// TwinCAT 3 PLC project ExternControl
// ProgramVersion: 3.1.4026.19
// libraries:
//   Tc2_Standard, * (Beckhoff Automation GmbH)
//   Tc2_System, * (Beckhoff Automation GmbH)
//   Tc2_Utilities, * (Beckhoff Automation GmbH)
//   VisuDialogs, * (System)
//   VisuDialogs
// project tree:
//   APPLICATION/ fb_Simulation.TcPOU (not stored), GVL_APPLICATION.TcGVL (not stored), MAIN_APP.TcPOU (not stored)
//   APPLICATION/_types/ E_PROCESS_CHECK.TcDUT (not stored), E_PROCESS_CTRL.TcDUT (not stored), E_PROCESS_STATE.TcDUT (not stored), ST_PROCESS_CTRL.TcDUT (not stored), ST_PROCESS_STATE.TcDUT (not stored), T_PROCESS.TcDUT (not stored)
//   APPLICATION/_types/fb_Instance/ E_INSTANCE_CHECK.TcDUT (not stored), E_INSTANCE_STATE.TcDUT (not stored), fb_Instance.TcPOU (not stored)
//   APPLICATION/_types/LinkedList/ fb_Process_LinkedListCtrl.TcPOU (not stored), I_Process_LinkedList.TcIO, ST_PROCESS_DATA.TcDUT (not stored), ST_PROCESS_LIST_RESULT.TcDUT (not stored)
//   / GlobalTextList.TcGTLO (not stored), MAIN.TcPOU, PlcTask.TcTTO (not stored), Visualization Manager.TcVMO (not stored)
//   MAPPING/ MAPPING_in.TcPOU, MAPPING_out.TcPOU
//   MAPPING/_types/ U_APP_CTRL.TcDUT (not stored), U_APP_STATE.TcDUT, U_INSTANCE_CTRL.TcDUT (not stored), U_INSTANCE_STATE.TcDUT (not stored), U_MOVER_CTRL.TcDUT, U_MOVER_INFO.TcDUT (not stored), U_MOVER_STATE.TcDUT (not stored), U_MOVE_DATA.TcDUT, U_TICKET_LIST_CTRL.TcDUT (not stored), U_TICKET_LIST_DATA_INPUT.TcDUT (not stored), U_TICKET_LIST_DATA_OUTPUT.TcDUT (not stored), U_TICKET_LIST_STATE.TcDUT, U_XTS_STATION_CTRL.TcDUT (not stored), U_XTS_STATION_STATE.TcDUT (not stored), U_XTS_TRANSPORT_CTRL.TcDUT (not stored), U_XTS_TRANSPORT_STATE.TcDUT (not stored)
//   MSG/ fb_LocalTime.TcPOU (not stored), fb_MessageData.TcPOU, fb_MessageDataCtrl.TcPOU (not stored), f_MessageSet.TcPOU (not stored), GVL_MSG.TcGVL, I_MessageData.TcIO
//   MSG/types/ e_Device.TcDUT (not stored), E_MessageType.TcDUT (not stored), E_MESSAGE_BATCH.TcDUT, E_MESSAGE_CHECK.TcDUT, E_MESSAGE_CTRL.TcDUT (not stored), E_MESSAGE_FLOW.TcDUT (not stored), E_MESSAGE_STATE.TcDUT (not stored), e_Subdevice.TcDUT (not stored), ST_Message.TcDUT (not stored), ST_MESSAGE_CTRL.TcDUT (not stored), ST_MESSAGE_STATE.TcDUT, TL_E_MESSAGETYPE.TcTLO (not stored)
//   XTS/CaGroup/types/ E_CA_GROUP_STATE.TcDUT (not stored), E_GROUP_CHECK.TcDUT (not stored), ST_GROUP_INFO.TcDUT (not stored)
//   XTS/ GVL_XTS.TcGVL, XTS_Parameter.TcGVL (not stored)
//   XTS/Mover/types/ E_MOVER_CTRL.TcDUT, E_MOVER_STATE.TcDUT (not stored), ST_GEAR_DATA.TcDUT (not stored), ST_MOVER_CTRL.TcDUT (not stored), ST_MOVER_INFO.TcDUT (not stored), ST_MOVER_STATE.TcDUT (not stored), ST_MOVE_DATA.TcDUT
//   XTS/Xpu/types/ E_XPU_CHECK.TcDUT (not stored), E_XPU_CTRL.TcDUT (not stored), E_XPU_INIT.TcDUT (not stored), E_XPU_STATE.TcDUT (not stored), ST_XPU_CTRL.TcDUT, ST_XPU_INFO.TcDUT (not stored), ST_XPU_STATE.TcDUT (not stored)
//   XTS/XtsStation/_types/ E_STATION_CTRL.TcDUT (not stored), E_STATION_GEAR_DISTANCE_AXIS.TcDUT (not stored), E_STATION_STATE.TcDUT (not stored), E_STATION_TYPE.TcDUT, ST_STATION_CTRL.TcDUT (not stored), ST_STATION_GEAR_PARAMETER.TcDUT, ST_STATION_LIST_RESULT.TcDUT (not stored), ST_STATION_MOVER_DATA.TcDUT (not stored), ST_STATION_PARAMETER.TcDUT (not stored), ST_STATION_STATE.TcDUT (not stored), T_NEST_OFFSET.TcDUT (not stored)
//   XTS/XtsTransportUnit/types/ E_XTS_TRANSPORT_CHECK.TcDUT (not stored), E_XTS_TRANSPORT_CTRL.TcDUT (not stored), E_XTS_TRANSPORT_STATE.TcDUT (not stored), ST_XTS_TRANSPORT_CTRL.TcDUT (not stored), ST_XTS_TRANSPORT_STATE.TcDUT (not stored)
//   XTS/_types/ E_PROGRESS.TcDUT (not stored), f_GetProgress.TcPOU (not stored), f_GetState.TcPOU
//   XTS/_Visualization/ GROUP_VISU.TcVIS, MOVER_VISU.TcVIS (not stored), STATION_VISU.TcVIS (not stored), XPU_VISU.TcVIS (not stored), XTS_TRANSPORT.TcVIS (not stored)
//   XTS/_Visualization/textlists/ TL_E_CTRL_MOVER.TcTLO, TL_E_CTRL_STATION.TcTLO (not stored), TL_E_CTRL_TRANSPORT.TcTLO (not stored), TL_E_CTRL_XPU.TcTLO (not stored)
//   XTS/_Visualization/types/ ST_XPU_STRINGS.TcDUT
// (motion and I/O tree: see PLC project xtstransport)
// real-time tasks:
//   TASK XTS Task 1: cycle T#250us, priority 1, ADS port 350
//   TASK PlcTask: cycle T#2ms, priority 15, ADS port 351
//   TASK Job Task: cycle default, priority 32
// variable links:
//   ExternControl/ExternControl Instance <-> XtsTransport/XtsTransport Instance
//     PlcTask Inputs/MAPPING_in.MoverInfo.byInfo <-> PlcTask Outputs/MAPPING_out.MoverInfo.byInfo
//     PlcTask Inputs/MAPPING_in.MoverState.byState <-> PlcTask Outputs/MAPPING_out.MoverState.byState
//     PlcTask Inputs/MAPPING_in.TransportState.byState <-> PlcTask Outputs/MAPPING_out.TransportState.byState
//     PlcTask Outputs/MAPPING_out.MoveData.byData <-> PlcTask Inputs/MAPPING_in.MoveData.byData
//     PlcTask Outputs/MAPPING_out.MoverControl.byCtrl <-> PlcTask Inputs/MAPPING_in.MoverCtrl.byCtrl
//     PlcTask Outputs/MAPPING_out.TransportControl.byCtrl <-> PlcTask Inputs/MAPPING_in.TransportControl.byCtrl

// ---- MAPPING/_types/U_APP_STATE.TcDUT
TYPE U_APP_STATE :
UNION
  stState             : ST_APP_STATE;
  byState   AT %i*    : ARRAY[1..SIZEOF(ST_APP_STATE)] OF BYTE;
END_UNION
END_TYPE

// ---- MAPPING/_types/U_MOVER_CTRL.TcDUT
TYPE U_MOVER_CTRL :
UNION
  stCtrl              : ARRAY[1..MAX_MOVER] OF ST_MOVER_CTRL;

  byCtrl    AT %Q*    : ARRAY[1..MAX_MOVER] OF
                        ARRAY[1..SIZEOF(ST_MOVER_CTRL)] OF BYTE;
END_UNION
END_TYPE

// ---- MAPPING/_types/U_MOVE_DATA.TcDUT
TYPE U_MOVE_DATA :
UNION
  stData              : ARRAY[1..MAX_MOVER] OF ST_MOVE_DATA;

  byData    AT %Q*    : ARRAY[1..MAX_MOVER] OF
                        ARRAY[1..SIZEOF(ST_MOVE_DATA)] OF BYTE;
END_UNION
END_TYPE

// ---- MAPPING/_types/U_TICKET_LIST_STATE.TcDUT
TYPE U_TICKET_LIST_STATE :
UNION
  stState             : ST_LIST_STATE;
  byState   AT %I*    : ARRAY[1..SIZEOF(ST_LIST_STATE)] OF BYTE;
END_UNION
END_TYPE

// ---- MSG/types/E_MESSAGE_BATCH.TcDUT
{attribute 'qualified_only'}
{attribute 'strict'}
{attribute 'to_string'}
TYPE E_MESSAGE_BATCH :
(
	MSG_BATCH_NULL,
  MSG_BATCH_JOB_STARTED,
  MSG_BATCH_NEXT_IN_JOB,
  MSG_BATCH_JOB_DONE
)UINT;
END_TYPE

// ---- MSG/types/E_MESSAGE_CHECK.TcDUT
{attribute 'qualified_only'}
{attribute 'strict'}
{attribute 'to_string'}
TYPE E_MESSAGE_CHECK :
(
  // 9000 --> here comes your error
  MSG_CHECK_INVALID_POINTER             := 9000,
  MSG_CHECK_INVALID_POINTER_TIME,
  MSG_CHECK_INVALID_POINTER_LIST,
  MSG_CHECK_INVALID_POINTER_MSG_IDX,
  MSG_CHECK_INVALID_POINTER_ERR_IDX,
  MSG_CHECK_INVALID_POINTER_ROOT_FILE,
  MSG_CHECK_INVALID_POINTER_ROOT_DIR,
  MSG_CHECK_INVALID_POINTER_CTRL,
  MSG_CHECK_INVALID_POINTER_STATE,

  // 10000 --> here comes your man
  MSG_CHECK_DONE                        := 10000
)UINT;
END_TYPE

// ---- MSG/types/ST_MESSAGE_STATE.TcDUT
TYPE ST_MESSAGE_STATE :
STRUCT
  State         : E_MESSAGE_STATE;  // as always... combined value of Cmd equivalent and e_progress
END_STRUCT
END_TYPE

// ---- XTS/Mover/types/E_MOVER_CTRL.TcDUT
{attribute 'qualified_only'}
{attribute 'strict'}
{attribute 'to_string'}
TYPE E_MOVER_CTRL :
(
  MOVER_NULL,               // initial value at startup, used for change of order or retrigger
  MOVER_ENABLE,             // sets MC_Power.Enable
  MOVER_DISABLE,            // removes MC_Power.Enable
  MOVER_MOVE_TO_POS,        // modulo absolute positioning with MC_MoveAbsolute, InTargetPosition check
  MOVER_MOVE_TO_POS_CA,     // modulo absolute positioning with MC_MoveAbsoluteCA, InTargetPosition check
  MOVER_SEND_TO_POS_CA,     // modulo absolute positioning with MC_MoveAbsoluteCA, done after moving ReleaseDistance
  MOVER_HALT,               // halts mover; by use of MC_Halt mover is set passive in CA group
  MOVER_GEAR_IN,            // GearIn for mover in standstill

  MOVER_GEAR_IN_POS_CA,     // GearInPosCA of mover; when FB_GearInPosCa is InSync --> order is done; check SyncDistance yourself and release mover with e_mover_order.mover_SendToPos
  MOVER_GEAR_OUT,           // gear out for mover
  MOVER_RESET,              // MC_RESET for mover
  MOVER_MOVE_TO_POS_ABS    // absolute positioning with MC_MoveAbsolute, InTargetPosition check
)UINT;
END_TYPE

// ---- XTS/Mover/types/ST_MOVE_DATA.TcDUT
{attribute 'pack_mode' := '2'}
TYPE ST_MOVE_DATA :
STRUCT
  // HAUD 2024 03 14
  // some init data added for example
  rPos            : LREAL :=   2275.0;
  rVelo           : LREAL :=    500.0;
  rAcc            : LREAL :=   5000.0;
  rJerk           : LREAL := 500000.0;
  rGap            : LREAL :=    100.0;
  rOverride       : LREAL :=    100.0;
  rDelta          : LREAL :=      0.05;
  rDistance       : LREAL :=     25.0;
END_STRUCT
END_TYPE

// ---- XTS/Xpu/types/ST_XPU_CTRL.TcDUT
{attribute 'pack_mode' := '2'}
TYPE ST_XPU_CTRL :
STRUCT
  Cmd             : E_XPU_CTRL;
END_STRUCT
END_TYPE

// ---- XTS/XtsStation/_types/E_STATION_TYPE.TcDUT
{attribute 'qualified_only'}
{attribute 'strict'}
{attribute 'to_string'}
TYPE E_STATION_TYPE :
(
	INVALID,
  STATION_PROCESS,      // default station with/without process
  STATION_GEAR_IN_POS   // GearInPos station for flying saw with MasterAxis
)USINT;
END_TYPE

// ---- XTS/XtsStation/_types/ST_STATION_GEAR_PARAMETER.TcDUT
TYPE ST_STATION_GEAR_PARAMETER :
STRUCT
  eDistance           : E_STATION_GEAR_DISTANCE_AXIS; // follow which leader?
  rSyncDistance       : LREAL := 100.0;               // synchrone distance while the mover is geared in
  rMinDistanceToSync  : LREAL := 100.0;               // minimum distance for mover to get nSync with the Master
END_STRUCT
END_TYPE

// ---- XTS/_Visualization/types/ST_XPU_STRINGS.TcDUT
TYPE ST_XPU_STRINGS :
STRUCT
  sXpuState       ,
  sXpuResult      ,
  sXpuCyclicCheck ,
  sXpuOpMode      ,
  sXpuMoverId_DetectionMode,
  sXpuMoverPosAssignement : STRING(30) := 'NULL';
END_STRUCT
END_TYPE

// ---- MSG/GVL_MSG.TcGVL
{attribute 'qualified_only'}
VAR_GLOBAL CONSTANT
  //-----------------------------------------------------------------------------
  // file paths for message system
  //  - compiler define option WIN switches to Windows file paths
  //-----------------------------------------------------------------------------
{IF defined (WIN)}
  {info 'WIN folders'}
  LOG_DIR               : STRING  := 'C:\TwinCAT\#MsgFiles\'; // delimiter at the end is mandatory!!
{ELSE}
  {info 'BSD folders'}
  LOG_DIR               : STRING  := '/usr/local/etc/TwinCAT/#MsgFiles/'; // delimiter at the end is mandatory!!
{END_IF}

  LOG_FILE              : STRING  := 'MSG_XtsTransport_';
  LOG_FILE_APP          : STRING  := 'MSG_Application_';
  LOG_FILE_METRIC       : STRING  := 'MSG_XtsTransportMetrics_';

  MAX_MESSAGE           : UINT    := 2000; // max entry in message list
END_VAR
VAR_GLOBAL
  //-----------------------------------------------------------------------------
  // Message System
  //  - Everybody uses f_MessageSet(ST_Message)
  //    - DECISION WHICH LIST IS MADE IN f_MessageSet !!
  //    - which list to use is determined by e_Device in your message
  //
  //  - MessageData instances are self sufficient and need only 
  //    datafield assignment for correct data-flow
  //
  //
  //-----------------------------------------------------------------------------
  //-----------------------------------------------------------------------------
  //-----------------------------------------------------------------------------
  // (ST_Message.eDevice := e_Device.Application)
  //----------------------------------------------------------------------------- 
  ApplicationMessageData          : fb_MessageDataCtrl;
  ApplicationMessageCtrl          : st_message_ctrl;
  ApplicationMessageState         : st_message_state;

  ApplicationMessages             : ARRAY[1..MAX_MESSAGE] OF ST_Message;
  MessageApplicationIndex         : UINT := 0; // message index for higher layers (grouping, Instances, etc.)
  MessageApplicationError         : UINT := 0; // error counter for higher learning
  //-----------------------------------------------------------------------------
  //-----------------------------------------------------------------------------
  // (ST_Message.eDevice := from Device_Null to XfcAxis)
  //-----------------------------------------------------------------------------
  TransportMessageData            : fb_MessageDataCtrl;
  TransportMessageCtrl            : st_message_ctrl;
  TransportMessageState           : st_message_state;

  TransportMessages               : ARRAY[1..MAX_MESSAGE] OF ST_Message;
  MessageTransportIndex           : UINT := 0; // message index for base layer
  MessageTransportError           : UINT := 0; // error counter for base layer
  //-----------------------------------------------------------------------------
  //-----------------------------------------------------------------------------
  // (ST_Message.eDevice := e_Device.Metrics)
  //-----------------------------------------------------------------------------
  MetricsMessageData              : fb_MessageDataCtrl;
  MetricsMessageCtrl              : st_message_ctrl;
  MetricsMessageState             : st_message_state;

  MetricsMessages                 : ARRAY[1..MAX_MESSAGE] OF ST_Message;
  MessageMetricsIndex             : UINT := 0; // message index for metrics data
  MessageMetricsError             : UINT := 0; // error counter for metrics data
  //-----------------------------------------------------------------------------
  //-----------------------------------------------------------------------------
  // (ST_Message.eDevice := e_Device.ProductData)
  //-----------------------------------------------------------------------------
  ProductMessageData              : fb_MessageDataCtrl;   // This is for you
  ProductMessageCtrl              : st_message_ctrl;
  ProductMessageState             : st_message_state;

  ProductMessages                 : ARRAY[1..MAX_MESSAGE] OF ST_Message;
  MessageProductIndex             : UINT := 0; // message index for your product data
  MessageProductError             : UINT := 0; // error counter for your product data
  //-----------------------------------------------------------------------------
  //-----------------------------------------------------------------------------
  fbLocalTime                     : fb_LocalTime;
  dtLocalTime                     : DT;
  sLocalTime                      : STRING;
  //-----------------------------------------------------------------------------
  //-----------------------------------------------------------------------------
  //-----------------------------------------------------------------------------
  //-----------------------------------------------------------------------------
  MessageLevelXpu                 : E_MessageType;
  MessageLevelStations            : ARRAY[1..MAX_STATION] OF E_MessageType;
  MessageLevelMovers              : ARRAY[1..MAX_MOVER]   OF E_MessageType;

  MessageLevelProcess             : ARRAY[1..MAX_PROCESS] OF E_MessageType;

{IF defined (TEST)}
  {info 'TEST logging enabled'}
  MessageLevel                    : E_MessageType := eMessageinfo; // a lot of messages
{ELSE}
  MessageLevel                    : E_MessageType := eMessageEmpty; // only errors are written into list 
{END_IF}

END_VAR

// ---- XTS/GVL_XTS.TcGVL
{attribute 'qualified_only'}
VAR_GLOBAL
  //---------------------------------------------------------------------------
  // XTS Station
  //  - handshakes mover in station with extern control
  //  - station parameters (positions, gap, dyn. constraints, description...)
//  StationStart        : ST_STATION_PARAMETER;   // Xts transport is sending all mover to this position (CMD_TRANSPORT_START)
//  StationStartIndex   : UINT := 1;              // index of XtsStation where all movers are entered into linked list.

  // station handshaking with mover and extern process
  // station sends mover to target station/WaitPos
  // station adds mover data to LinkedList.AddTail() of target station
//  Station             : ARRAY[1..MAX_STATION] OF fb_StationProcess;
//  StationGearIn       : ARRAY[1..MAX_STATION] OF fb_StationGearInPos;
//
//  StationList         : ARRAY[1..MAX_STATION] OF fb_Station_LinkedList;
//
//  StationQueue        : ARRAY[1..MAX_STATION]    OF 
//                        ARRAY[1..MAX_LIST_NODES] OF ST_STATION_MOVER_DATA;
//
//  // interface for access to List methods
//  StationListItf      : ARRAY[1..MAX_STATION] OF I_Station_LinkedList;
//
//  // interface for access to station methods
//  StationCtrlItf      : ARRAY[1..MAX_STATION] OF I_XtsTransport_Station;

  // ctrl / state datafields for extern control
  StationCtrl         : ARRAY[1..MAX_STATION] OF ST_STATION_CTRL;   // control for extern to write, you can do whatever you want as long as you do as I say
  StationState        : ARRAY[1..MAX_STATION] OF ST_STATION_STATE;  // state for extern to read, this is what I tell you to do

  // station parameter
//  StationParameter    : ARRAY[1..MAX_STATION] OF ST_STATION_PARAMETER; // wherever, whenever you want. Build it and they will come...

  // station GearInPosCA parameter and data structs
//  StationGearParameter: ARRAY[1..MAX_STATION] OF ST_STATION_GEAR_PARAMETER;
//  StationGearData     : ARRAY[1..MAX_STATION] OF ST_GEAR_DATA;

  // static position offsets in stations
//  PositionOffset      : ARRAY[1..MAX_STATION] OF T_NEST_OFFSET; // added to PosStop[] in XtsStation


  //---------------------------------------------------------------------------
  // XTS
  // XTS TransportUnit
  //  - This is ground control
  //  - handles request for XPU, Group, Mover, StartUp, ReStart
//  XtsTransport        : fb_TransportUnit;         // manages members of XTS transport for extern to access

  XtsTransportCtrl    : ST_XTS_TRANSPORT_CTRL;    // control of XTS transport for extern to write
  XtsTransportState   : ST_XTS_TRANSPORT_STATE;   // state   of XTS transport for extern to read


  //---------------------------------------------------------------------------
  // XPU
  // XTS-Utility checks
  // XTS-Utility interfaces for you to use
//  Xpu             : fb_XpuCtrl;

//  XpuCtrl         : ST_XPU_CTRL;
//  XpuState        : ST_XPU_STATE;
//  XpuInfo         : ST_XPU_INFO;
//  XpuModules      : ARRAY[1..MAX_MODULE] OF Tc3_XTS_Utility.ST_InfoDataView;


  //---------------------------------------------------------------------------
  // Collision avoidance group CA
  //
  // - add mover to group
  // - build group
  // - clear group
  // - whereever you may roam, no on will tread on you
//  CaGroup         : FB_CaGroup;                   // cyclic check of CaGroup state and errors; carries methods for handling CaGroup
//  CaGroupItf      : I_XtsTransport_CaGroup;       // Interface used by fb_TransportUnit

  // cyclic mapping to MOTION/Objects/CaGroup 
//  CaGroupRef      : Tc3_McCoordinatedMotion.AXES_GROUP_REF;

  // Info data from CaGroup FB
//  CaGroupInfo     : ST_GROUP_INFO;                // cyclic info about CaGroup for fb_TransportUnit to read
  //---------------------------------------------------------------------------

  //---------------------------------------------------------------------------
  // MC2 encapsulation, CA movement
//  Mover           : ARRAY[1..MAX_MOVER] OF fb_MoverCtrl;    // MC and CA methods for mover; cyclic check for individual command on mover

  MoverCtrl       : ARRAY[1..MAX_MOVER] OF ST_MOVER_CTRL;   // control of individual mover for extern to write
  MoverState      : ARRAY[1..MAX_MOVER] OF ST_MOVER_STATE;  // state   of individual mover for extern to read

//  MoverItf        : ARRAY[1..MAX_MOVER] OF I_XtsTransport_Mover;  // Interface used by fb_TransportUnit

//  LastPosition    : ARRAY[1..MAX_MOVER] OF LREAL;           // on execute of any movement, value is saved here (used by fb_Mover)
//  LastGap         : ARRAY[1..MAX_MOVER] OF LREAL;           // on execute of any movement, value is saved here (used by fb_Mover)

  MoverInfo       : ARRAY[1..MAX_MOVER] OF ST_MOVER_INFO;   // cyclic info about mover for extern to read

  MoveData        : ARRAY[1..MAX_MOVER] OF ST_MOVE_DATA;    // dynamic constraints for move commands
  GearData        : ARRAY[1..MAX_MOVER] OF ST_GEAR_DATA;    // dynamic constraints and positions for GearIn/GearInPosCa
  
  // cyclic mapping to MOTION/Axes
//  AxisRefMover    : ARRAY[1..MAX_MOVER] OF Tc2_MC2.AXIS_REF;
  //---------------------------------------------------------------------------
END_VAR

// ---- APPLICATION/_types/LinkedList/I_Process_LinkedList.TcIO
INTERFACE I_Process_LinkedList

METHOD AddHeadValue : ST_PROCESS_LIST_RESULT
VAR_INPUT
  stData        : ST_PROCESS_DATA;
END_VAR
END_METHOD

METHOD AddTailValue : ST_PROCESS_LIST_RESULT
VAR_INPUT
  stData        : ST_PROCESS_DATA;
END_VAR
END_METHOD

PROPERTY Count : UDINT
GET
END_GET
END_PROPERTY

PROPERTY Data : ARRAY[1..MAX_LIST_NODES] OF ST_PROCESS_DATA
GET
END_GET
END_PROPERTY

PROPERTY Free : UDINT
GET
END_GET
END_PROPERTY

METHOD GetHead : ST_PROCESS_LIST_RESULT
VAR_INPUT
END_VAR
END_METHOD

METHOD InitList : BOOL
END_METHOD

PROPERTY Nodes : ARRAY[0..MAX_LIST_NODES] OF T_LinkedListEntry
GET
END_GET
END_PROPERTY

METHOD RemoveHeadValue : ST_PROCESS_LIST_RESULT
VAR_INPUT
END_VAR
END_METHOD

END_INTERFACE

// ---- MSG/I_MessageData.TcIO
INTERFACE I_MessageData

PROPERTY DirRoot : POINTER to string(255)
SET
END_SET
END_PROPERTY

PROPERTY ErrorIndex : reference to uint
SET
END_SET
END_PROPERTY

PROPERTY FileRoot : pointer to string(255)
SET
END_SET
END_PROPERTY

PROPERTY LocalTime : pointer to DT
SET
END_SET
END_PROPERTY

PROPERTY MessageIndex : reference to uint
SET
END_SET
END_PROPERTY

PROPERTY MsgList : pointer to ARRAY[1..GVL_MSG.MAX_MESSAGE] OF st_message
SET
END_SET
END_PROPERTY

END_INTERFACE

// ---- MAIN.TcPOU
//---------------------------------------------------------------------------------------------------------------
//
//  HAUD 2026.01.16
//
//  - ExternControl
//
//    - placeholder programm for specific implementation of machine logic
//
//---------------------------------------------------------------------------------------------------------------
PROGRAM MAIN
VAR
	bInit 				          : BOOL;
  eInit                   : E_PROGRESS := E_PROGRESS.PROGRESS_DONE; // empty right now, so init is done

  nStation,
	nMover,
  nMoverSelected,
  nStationSelected,
  nStationParameter       : UINT;

  sStationText            : STRING(30);
  stXpuStrings            : ST_XPU_STRINGS;

  eTransportState         : E_XTS_TRANSPORT_STATE;
  eTransportResult        : E_PROGRESS;

  eXpuState               : E_XPU_STATE;
  eXpuResult              : E_PROGRESS;
  eXpuCheck               : E_XPU_CHECK;

  eMoverState             : E_MOVER_STATE;
  eMoverResult            : E_PROGRESS;

  sCaGroupState,
  sTransportState,
  sTransportCheck,
  sTransportResult,
  sMoverState,
  sMoverResult,
  sStationState,
  sStationStateMask,
  sStationCtrlMask        : STRING;

  bStationEnable,
  bStationEnter,
  bStationStart,
  bStationDone,
  bStationOut,
  bStationGone            : BOOL;

  nStn                    : UINT;

  stMsg                   : ST_Message;
  eMsgState               : e_message_state;
  eMsgProgress            : E_PROGRESS;
  eMtrState               : e_message_state;
  eMtrProgress            : E_PROGRESS;

  bGetVariant             : BOOL := TRUE;
  nVariant                : UINT;

  rGap                    : REAL :=     105.0;
  rAcc                    : REAL :=  17_500.0;
  rJerk                   : REAL := 600_000.0;
END_VAR

//############################################################################
//############################################################################
//  /Visualization data	
//############################################################################
VisualizationData();
//############################################################################
//  Visualization data/	
//############################################################################

ACTION VisualizationData:
//############################################################################
//############################################################################
// Visualization data	
//############################################################################
// get enumerations from XPU for visu:	
eTransportState                       := f_GetState   (GVL_XTS.XtsTransportState.State);
eTransportResult                      := f_GetProgress(GVL_XTS.XtsTransportState.State);

eXpuState                             := f_GetState   (GVL_XTS.XtsTransportState.XpuState.State);
eXpuResult                            := f_GetProgress(GVL_XTS.XtsTransportState.XpuState.State);

eXpuCheck                             := GVL_XTS.XtsTransportState.XpuState.Check;

// display xpu state and result in visu
// get strings and info
sCaGroupState                         := TO_STRING(GVL_XTS.XtsTransportState.GroupInfo.CaGroupState);

sTransportState                       := TO_STRING(eTransportState);
sTransportCheck                       := TO_STRING(GVL_XTS.XtsTransportState.Check);
sTransportResult                      := TO_STRING(eTransportResult);

stXpuStrings.sXpuState                := TO_STRING(eXpuState);
stXpuStrings.sXpuResult               := TO_STRING(eXpuResult);
stXpuStrings.sXpuCyclicCheck          := TO_STRING(eXpuCheck);

stXpuStrings.sXpuOpMode               := TO_STRING(GVL_XTS.XtsTransportState.XpuInfo.OperationMode);
stXpuStrings.sXpuMoverId_DetectionMode:= TO_STRING(GVL_XTS.XtsTransportState.XpuInfo.IdDetectionMode);
stXpuStrings.sXpuMoverPosAssignement  := TO_STRING(GVL_XTS.XtsTransportState.XpuInfo.MoverPositionAssignement);

nMoverSelected                        := SEL((nMoverSelected<1), nMoverSelected, 1);
nMoverSelected                        := SEL((nMoverSelected>MAX_MOVER), nMoverSelected, MAX_MOVER);

nStationSelected                      := SEL((nStationSelected<1), nStationSelected, 1);
nStationSelected                      := SEL((nStationSelected>MAX_STATION), nStationSelected, MAX_STATION);

//bStationEnable                        := SEL((GVL_XTS.StationCtrl[nStationSelected].Cmd = E_STATION_CTRL.STATION_ENABLE),        FALSE, TRUE);
//bStationEnter                         := SEL((GVL_XTS.StationCtrl[nStationSelected].Cmd = E_STATION_CTRL.STATION_MOVER_ENTER),   FALSE, TRUE);
//bStationStart                         := SEL((GVL_XTS.StationCtrl[nStationSelected].Cmd = E_STATION_CTRL.STATION_PROCESS_START), FALSE, TRUE);
//bStationDone                          := SEL((GVL_XTS.StationCtrl[nStationSelected].Cmd = E_STATION_CTRL.STATION_PROCESS_DONE),  FALSE, TRUE);
//bStationOut                           := SEL((GVL_XTS.StationCtrl[nStationSelected].Cmd = E_STATION_CTRL.STATION_MOVER_OUT),     FALSE, TRUE);
//bStationGone                          := SEL((GVL_XTS.StationCtrl[nStationSelected].Cmd = E_STATION_CTRL.STATION_MOVER_GONE),    FALSE, TRUE);

eMoverState                           := f_GetState   (GVL_XTS.MoverState[nMoverSelected].State);
eMoverResult                          := f_GetProgress(GVL_XTS.MoverState[nMoverSelected].State);

sMoverState                           := TO_STRING(eMoverState);
sMoverResult                          := TO_STRING(eMoverResult);

//sStationState                         := TO_STRING(GVL_XTS.StationState[nStationSelected].State);
//sStationStateMask                     := Tc2_Utilities.BYTE_TO_BINSTR(GVL_XTS.StationState[nStationSelected].nMask, 8);
//sStationCtrlMask                      := Tc2_Utilities.BYTE_TO_BINSTR(GVL_XTS.StationCtrl[nStationSelected].nMask, 8);

//############################################################################
//############################################################################
END_ACTION

END_PROGRAM

// ---- XTS/_types/f_GetState.TcPOU
// global function to extract state identifier from combined value
FUNCTION f_GetState : uint
VAR_INPUT
  state     : UINT; // combined value of identifier + e_progress
END_VAR
VAR
  _stx      : uint;
END_VAR

_stx          := state MOD E_PROGRESS.PROGRESS_INIT;

IF (_stx = 0)
THEN
  f_GetState  := state;
ELSE
  f_GetState  := _stx;
END_IF

END_FUNCTION

// ---- MAPPING/MAPPING_in.TcPOU
PROGRAM MAPPING_in
VAR
  sMapping          : STRING;
  bFirstCycle       : BOOL := TRUE;



//  TicketListOutput  : U_TICKET_LIST_DATA_OUTPUT;
//  TicketListState   : U_TICKET_LIST_STATE;
//  InstanceState     : U_INSTANCE_STATE;
//  AppState          : U_APP_STATE;
  TransportState    : U_XTS_TRANSPORT_STATE;
  StationState      : U_XTS_STATION_STATE;
  MoverState        : U_MOVER_STATE;
  MoverInfo         : U_MOVER_INFO;

  szTransportState  : ARRAY[1..2] OF UDINT;
  szStationState    : ARRAY[1..2] OF UDINT;
  szMoverState      : ARRAY[1..2] OF UDINT;
  szMoverInfo       : ARRAY[1..2] OF UDINT;

  szAppState        : ARRAY[1..2] OF UDINT;
  szInstanceState   : ARRAY[1..2] OF UDINT;
  szTicketState     : ARRAY[1..2] OF UDINT;
  szTicketData      : ARRAY[1..2] OF UDINT;
END_VAR


IF (bFirstCycle)
THEN
  bFirstCycle           := FALSE;
  
  szTransportState[1]   := SIZEOF(TransportState);
  szTransportState[2]   := SIZEOF(GVL_XTS.XtsTransportState);

  szStationState  [1]   := SIZEOF(StationState);
  szStationState  [2]   := SIZEOF(GVL_XTS.StationState);

  szMoverState    [1]   := SIZEOF(MoverState);
  szMoverState    [2]   := SIZEOF(GVL_XTS.MoverState);

  szMoverInfo     [1]   := SIZEOF(MoverInfo);
  szMoverInfo     [2]   := SIZEOF(GVL_XTS.MoverInfo);


(*
  szAppState[1]       := SIZEOF(AppState);
  szAppState[2]       := SIZEOF(GVL_APPLICATION.AppState);

  szInstanceState[1]  := SIZEOF(InstanceState);
  szInstanceState[2]  := SIZEOF(GVL_APPLICATION.InstanceState);

  szTicketState[1]    := SIZEOF(TicketListState);
  szTicketState[2]    := SIZEOF(GVL_APPLICATION.TicketListState);

  szTicketData[1]     := SIZEOF(TicketListOutput);
  szTicketData[2]     := SIZEOF(GVL_APPLICATION.TicketListDataOutput);
*)
END_IF
(*
//---------------------------------------------------------------------
IF (SIZEOF(TicketListOutput) <> SIZEOF(GVL_APPLICATION.TicketListDataOutput))
THEN
  sMapping  := 'TicketListOutput sizes DO NOT match';
  RETURN;
END_IF
//---------------------------------------------------------------------
IF (SIZEOF(TicketListState) <> SIZEOF(GVL_APPLICATION.TicketListState))
THEN
  sMapping  := 'TicketListState sizes DO NOT match';
  RETURN;
END_IF
//---------------------------------------------------------------------
IF (SIZEOF(InstanceState) <> SIZEOF(GVL_APPLICATION.InstanceState))
THEN
  sMapping  := 'InstanceState sizes DO NOT match';
  RETURN;
END_IF
//---------------------------------------------------------------------
IF (SIZEOF(AppState) <> SIZEOF(GVL_APPLICATION.AppState))
THEN
  sMapping  := 'AppState sizes DO NOT match';
  RETURN;
END_IF
*)
//---------------------------------------------------------------------
IF (SIZEOF(TransportState) <> SIZEOF(GVL_XTS.XtsTransportState))
THEN
  sMapping  := 'TransportState sizes DO NOT match';
  RETURN;
END_IF
//---------------------------------------------------------------------
IF (SIZEOF(StationState) <> SIZEOF(GVL_XTS.StationState))
THEN
  sMapping  := 'StationState sizes DO NOT match';
  RETURN;
END_IF
IF (SIZEOF(MoverState) <> SIZEOF(GVL_XTS.MoverState))
THEN
  sMapping  := 'MoverState sizes DO NOT match';
  RETURN;
END_IF
IF (SIZEOF(MoverInfo) <> SIZEOF(GVL_XTS.MoverInfo))
THEN
  sMapping  := 'MoverInfo sizes DO NOT match';
  RETURN;
END_IF
sMapping    := 'MAPPING ACTIVE';
//-----------------------------------------------------------------------------------------
//       destination,                               source,                size
//-----------------------------------------------------------------------------------------
  memcpy(ADR(GVL_XTS.XtsTransportState),            ADR(TransportState),  SIZEOF(TransportState));
  memcpy(ADR(GVL_XTS.StationState),                 ADR(StationState),    SIZEOF(StationState));
  memcpy(ADR(GVL_XTS.MoverState),                   ADR(MoverState),      SIZEOF(MoverState));
  memcpy(ADR(GVL_XTS.MoverInfo),                    ADR(MoverInfo),       SIZEOF(MoverInfo));

  //memcpy(ADR(GVL_APPLICATION.AppState),             ADR(AppState),         SIZEOF(AppState));
  //GVL_APPLICATION.AppState.AppInit                  := AppSTate.stState.AppInit;

  //memcpy(ADR(GVL_APPLICATION.InstanceState),        ADR(InstanceState),    SIZEOF(InstanceState));
  //memcpy(ADR(GVL_APPLICATION.TicketListState),      ADR(TicketListState),  SIZEOF(TicketListState));
  //memcpy(ADR(GVL_APPLICATION.TicketListDataOutput), ADR(TicketListOutput), SIZEOF(TicketListOutput));
//-----------------------------------------------------------------------------------------
//-----------------------------------------------------------------------------------------

END_PROGRAM

// ---- MAPPING/MAPPING_out.TcPOU
PROGRAM MAPPING_out
VAR
  sMapping          : STRING;

  bFirstCycle       : BOOL := TRUE;

//  TicketListInput   : U_TICKET_LIST_DATA_INPUT;
//  TicketListControl : U_TICKET_LIST_CTRL;
//  InstanceCtrl      : U_INSTANCE_CTRL;
//  AppControl        : U_APP_CTRL;
  TransportControl  : U_XTS_TRANSPORT_CTRL;
  StationControl    : U_XTS_STATION_CTRL;
  MoverControl      : U_MOVER_CTRL;
  MoveData          : U_MOVE_DATA;



  szTransportCtrl   : ARRAY[1..2] OF UDINT;
  szStationControl  : ARRAY[1..2] OF UDINT;
  szMoverControl    : ARRAY[1..2] OF UDINT;
  szMoveData        : ARRAY[1..2] OF UDINT;

  szAppCtrl         : ARRAY[1..2] OF UDINT;
  szInstanceCtrl    : ARRAY[1..2] OF UDINT;
  szTicketCtrl      : ARRAY[1..2] OF UDINT;
  szTicketData      : ARRAY[1..2] OF UDINT;
END_VAR


IF (bFirstCycle)
THEN
  bFirstCycle             := FALSE;

  szTransportCtrl[1]      := SIZEOF(TransportControl);
  szTransportCtrl[2]      := SIZEOF(GVL_XTS.XtsTransportCtrl);

  szStationControl[1]     := SIZEOF(StationControl);
  szStationControl[2]     := SIZEOF(GVL_XTS.StationCtrl);

  szMoverControl[1]       := SIZEOF(MoverControl);
  szMoverControl[2]       := SIZEOF(GVL_XTS.MoverCtrl);

  szMoveData    [1]       := SIZEOF(MoveData);
  szMoveData    [2]       := SIZEOF(GVL_XTS.MoveData);

(*
  szAppCtrl  [1]          := SIZEOF(AppControl);
  szAppCtrl  [2]          := SIZEOF(GVL_APPLICATION.AppControl);

  szInstanceCtrl [1]      := SIZEOF(MAPPING_out.InstanceCtrl);
  szInstanceCtrl [2]      := SIZEOF(MAPPING_out.InstanceCtrl);

  szTicketCtrl[1]         := SIZEOF(TicketListControl);
  szTicketCtrl[2]         := SIZEOF(GVL_APPLICATION.TicketListControl);

  szTicketData[1]         := SIZEOF(TicketListInput);
  szTicketData[2]         := SIZEOF(GVL_APPLICATION.TicketListDataInput);
*)
END_IF
(*
//---------------------------------------------------------------------
IF (SIZEOF(TicketListInput) <> SIZEOF(GVL_APPLICATION.TicketListDataInput))
THEN
  sMapping  := 'TicketListInput sizes DO NOT match';
  RETURN;
END_IF
//---------------------------------------------------------------------
IF (SIZEOF(TicketListControl) <> SIZEOF(GVL_APPLICATION.TicketListControl))
THEN
  sMapping  := 'TicketListControl sizes DO NOT match';
  RETURN;
END_IF
//---------------------------------------------------------------------
IF (SIZEOF(InstanceCtrl) <> SIZEOF(GVL_APPLICATION.InstanceCtrl))
THEN
  sMapping  := 'InstanceCtrl sizes DO NOT match';
  RETURN;
END_IF
//---------------------------------------------------------------------
IF (SIZEOF(AppControl) <> SIZEOF(GVL_APPLICATION.AppControl))
THEN
  sMapping  := 'AppControl sizes DO NOT match';
  RETURN;
END_IF
*)
//---------------------------------------------------------------------
IF (SIZEOF(TransportControl) <> SIZEOF(GVL_XTS.XtsTransportCtrl))
THEN
  sMapping  := 'TransportControl sizes DO NOT match';
  RETURN;
END_IF
IF (SIZEOF(StationControl) <> SIZEOF(GVL_XTS.StationCtrl))
THEN
  sMapping  := 'StationControl sizes DO NOT match';
  RETURN;
END_IF
IF (SIZEOF(MoverControl) <> SIZEOF(GVL_XTS.MoverCtrl))
THEN
  sMapping  := 'MoverControl sizes DO NOT match';
  RETURN;
END_IF
IF (SIZEOF(MoveData) <> SIZEOF(GVL_XTS.MoveData))
THEN
  sMapping  := 'MoveData sizes DO NOT match';
  RETURN;
END_IF
sMapping    := 'MAPPING_OUTPUT_ACTIVE';
//---------------------------------------------------------------------
//       destination,                       source,                size
//---------------------------------------------------------------------
  memcpy(ADR(TransportControl), ADR(GVL_XTS.XtsTransportCtrl),       SIZEOF(TransportControl));
  memcpy(ADR(StationControl),   ADR(GVL_XTS.StationCtrl),            SIZEOF(StationControl));
  memcpy(ADR(MoverControl),     ADR(GVL_XTS.MoverCtrl),              SIZEOF(MoverControl));
  memcpy(ADR(MoveData),         ADR(GVL_XTS.MoveData),               SIZEOF(MoveData));

//  memcpy(ADR(AppControl),       ADR(GVL_APPLICATION.AppControl),          SIZEOF(AppControl));
//  memcpy(ADR(InstanceCtrl),     ADR(GVL_APPLICATION.InstanceCtrl),        SIZEOF(InstanceCtrl));
//  memcpy(ADR(TicketListControl),ADR(GVL_APPLICATION.TicketListControl),   SIZEOF(TicketListControl));
//  memcpy(ADR(TicketListInput),  ADR(GVL_APPLICATION.TicketListDataInput), SIZEOF(TicketListInput));
//---------------------------------------------------------------------
//---------------------------------------------------------------------

END_PROGRAM

// ---- MSG/fb_MessageData.TcPOU
FUNCTION_BLOCK ABSTRACT fb_MessageData IMPLEMENTS I_MessageData
VAR CONSTANT
{attribute 'hide'}
  STR_LEN       : UDINT := 524_288;
END_VAR
VAR
  _eCheck       : E_MESSAGE_CHECK;            // pointer check state

  _pFileRoot    : POINTER TO STRING(255);     // you decide (example in GVL_MSG.LOG_FILE)
  _pDirRoot     : POINTER TO STRING(255);     // see GVL_MSG.LOG_DIR

  _nMsgIndex    : REFERENCE TO UINT;          // Hypnos IS the only one in the village, if there are more you need more villages
  _nErrIndex    : REFERENCE TO UINT;          // Thanatos, Hypnos stern and more serious brother

  _dtLocalTime  : POINTER TO DT;
  _pMsgList     : POINTER TO ARRAY[1..GVL_MSG.MAX_MESSAGE] OF ST_Message; // attach your list here

	_rtrigReset   : Tc2_Standard.R_TRIG;
	_aWriteList   : ARRAY[1..GVL_MSG.MAX_MESSAGE] OF ST_Message;
	_sWriteData   : STRING(STR_LEN);
	_sNewLine     : STRING := '$N';
	_sTab         : STRING := '$T';
	_iCount, 
	_iStart, 
	_iEnd         : UINT;

	_fbCreateDir  : Tc2_System.FB_CreateDir;
	_sTmp         : STRING(256);
	_sFilename    : STRING(256);
	_sFolderDate  : STRING;
	_bFileCreated : BOOL;

	_fbFileOpen   : Tc2_System.FB_FileOpen;
	_fbFileWrite  : Tc2_System.FB_FileWrite;
	_fbFileClose  : Tc2_System.FB_FileClose;
END_VAR

METHOD Builder : BOOL // string concat for length > 255
VAR_INPUT
  pInString   : POINTER TO STRING;
  pOutString  : POINTER TO STRING(STR_LEN);
  Length      : UINT;
END_VAR
VAR
  Counter     : UDINT;
  pInWork     : POINTER TO BYTE;
  pOutWork    : POINTER TO BYTE;
END_VAR
pOutWork := pOutString;
pInWork := pInString;
Counter := 0;

(*check termination*)
WHILE (pOutWork^ <> 0) AND
      (Counter < STR_LEN+1)
DO
  Counter := Counter + 1;
  pOutWork := pOutWork + 1;
END_WHILE

(* append only if data fits into output *)
IF (Counter + Length < STR_LEN+1)
THEN

  (* append data *)
  FOR Counter := 1 TO Length
  DO
    pOutWork^ := pInWork^;
    pOutWork := pOutWork + 1;
    pInWork := pInWork + 1;
  END_FOR

  (* terminate *)
  pOutWork := pOutWork + 1;
  pOutWork^ := 0;
END_IF
END_METHOD

METHOD Check : BOOL
VAR_INPUT
END_VAR

IF NOT (_dtLocalTime <> 0)
THEN
  _eCheck       := E_MESSAGE_CHECK.MSG_CHECK_INVALID_POINTER_TIME;
  RETURN;
END_IF

IF NOT (_pMsgList <> 0)
THEN
  _eCheck       := E_MESSAGE_CHECK.MSG_CHECK_INVALID_POINTER_LIST;
  RETURN;
END_IF

IF NOT (_pFileRoot <> 0)
THEN
  _eCheck       := E_MESSAGE_CHECK.MSG_CHECK_INVALID_POINTER_ROOT_FILE;
  RETURN;
END_IF

IF NOT (_pDirRoot <> 0)
THEN
  _eCheck       := E_MESSAGE_CHECK.MSG_CHECK_INVALID_POINTER_ROOT_DIR;
  RETURN;
END_IF

IF NOT __ISVALIDREF(_nMsgIndex)
THEN
  _eCheck       := E_MESSAGE_CHECK.MSG_CHECK_INVALID_POINTER_MSG_IDX;
  RETURN;
END_IF

IF NOT __ISVALIDREF(_nErrIndex)
THEN
  _eCheck       := E_MESSAGE_CHECK.MSG_CHECK_INVALID_POINTER_ERR_IDX;
  RETURN;
END_IF


_eCheck         := E_MESSAGE_CHECK.MSG_CHECK_DONE;
Check           := TRUE;
END_METHOD

METHOD Device_to_String : string
VAR_INPUT
  eMsgDevice    : e_Device;
END_VAR
VAR
  sId                 : STRING := '_ID_';
  nId                 : UDINT;
END_VAR
IF (eMsgDevice < e_device.General)
THEN
  // below general case
  nId := TO_UDINT(eMsgDevice);
  sId := concat(sId, TO_STRING(nId));

  Device_to_String := concat(TO_STRING(eMsgDevice), sId);

ELSE
  IF (eMsgDevice >= e_Device.DataProduct)
  THEN
    nId := eMsgDevice MOD e_Device.DataProduct;
    sId := concat(sId, TO_STRING(nId));
 
    Device_to_String := concat(TO_STRING(e_Device.DataProduct), sId);

  ELSIF (eMsgDevice >= e_Device.Application)
  THEN
    nId := eMsgDevice MOD e_Device.Application;
    sId := concat(sId, TO_STRING(nId));
 
    Device_to_String := concat(TO_STRING(e_Device.Application), sId);

  ELSIF (eMsgDevice >= e_Device.Process)
  THEN
    nId := eMsgDevice MOD e_Device.Process;
    sId := concat(sId, TO_STRING(nId));
 
    Device_to_String := concat(TO_STRING(e_Device.Process), sId);

  ELSIF (eMsgDevice >= e_Device.Metrics)
  THEN
    nId := eMsgDevice MOD e_Device.Metrics;
    sId := concat(sId, TO_STRING(nId));
 
    Device_to_String := concat(TO_STRING(e_device.Metrics), sId);

  ELSIF (eMsgDevice >= e_device.XfcAxis)
  THEN
    nId := eMsgDevice MOD e_device.XfcAxis;
    sId := concat(sId, TO_STRING(nId));
 
    Device_to_String := concat(TO_STRING(e_device.XfcAxis), sId);

  ELSIF (eMsgDevice >= e_device.Axis)
  THEN
    nId := eMsgDevice MOD e_device.Axis;
    sId := concat(sId, TO_STRING(nId));
 
    Device_to_String := concat(TO_STRING(e_device.Axis), sId);

  ELSIF (eMsgDevice >= e_device.NciChannelCtrl)
  THEN
    nId := eMsgDevice MOD e_device.NciChannelCtrl;
    sId := concat(sId, TO_STRING(nId));
 
    Device_to_String := concat(TO_STRING(e_device.NciChannelCtrl), sId);

  ELSIF (eMsgDevice >= e_device.NciChannel)
  THEN
    nId := eMsgDevice MOD e_device.NciChannel;
    sId := concat(sId, TO_STRING(nId));
 
    Device_to_String := concat(TO_STRING(e_device.NciChannel), sId);

  ELSIF (eMsgDevice >= e_Device.Camming)
  THEN
    nId := eMsgDevice MOD e_Device.Camming;
    sId := concat(sId, TO_STRING(nId));
 
    Device_to_String := concat(TO_STRING(e_device.Camming), sId);

  ELSIF (eMsgDevice >= e_Device.XtsStation)
  THEN
    nId := eMsgDevice MOD e_Device.XtsStation;
    sId := concat(sId, TO_STRING(nId));
 
    Device_to_String := concat(TO_STRING(e_device.XtsStation), sId);

  ELSIF (eMsgDevice >= e_Device.XfcTouchProbe)
  THEN
    nId := eMsgDevice MOD e_Device.XfcTouchProbe;
    sId := concat(sId, TO_STRING(nId));
 
    Device_to_String := concat(TO_STRING(e_device.XfcTouchProbe), sId);

  ELSIF (eMsgDevice >= e_Device.XfcTriggerBox)
  THEN
    nId := eMsgDevice MOD e_Device.XfcTriggerBox;
    sId := concat(sId, TO_STRING(nId));
 
    Device_to_String := concat(TO_STRING(e_device.XfcTriggerBox), sId);

  ELSIF (eMsgDevice >= e_Device.XtsTransportUnit)
  THEN
    nId := eMsgDevice MOD e_Device.XtsTransportUnit;
    sId := concat(sId, TO_STRING(nId));
 
    Device_to_String := concat(TO_STRING(e_device.XtsTransportUnit), sId);

  ELSIF (eMsgDevice >= e_Device.MoverCtrl)
  THEN
    nId := eMsgDevice MOD e_Device.MoverCtrl;
    sId := concat(sId, TO_STRING(nId));
 
    Device_to_String := concat(TO_STRING(e_device.MoverCtrl), sId);

  ELSIF (eMsgDevice >= e_Device.Mover)
  THEN
    nId := eMsgDevice MOD e_Device.Mover;
    sId := concat(sId, TO_STRING(nId));
 
    Device_to_String := concat(TO_STRING(e_device.Mover), sId);

  ELSIF (eMsgDevice >= e_Device.XpuCtrl)
  THEN
    nId := eMsgDevice MOD e_Device.XpuCtrl;
    sId := concat(sId, TO_STRING(nId));
 
    Device_to_String := concat(TO_STRING(e_device.XpuCtrl), sId);

  ELSIF (eMsgDevice >= e_Device.Xpu)
  THEN
    nId := eMsgDevice MOD e_Device.Xpu;
    sId := concat(sId, TO_STRING(nId));
 
    Device_to_String := concat(TO_STRING(e_device.Xpu), sId);

  ELSIF (eMsgDevice >= e_Device.CaGroup)
  THEN
    nId := eMsgDevice MOD e_Device.CaGroup;
    sId := concat(sId, TO_STRING(nId));
 
    Device_to_String := concat(TO_STRING(e_device.CaGroup), sId);

  ELSIF (eMsgDevice >= e_Device.General)
  THEN
    nId := eMsgDevice MOD e_Device.General;
    sId := concat(sId, TO_STRING(nId));
 
    Device_to_String := concat(TO_STRING(e_device.General), sId);

  ELSE
    Device_to_String := TO_STRING(eMsgDevice);
  END_IF
END_IF
END_METHOD

PROPERTY DirRoot : POINTER to string(255)
SET
_pDirRoot := DirRoot;
END_SET
END_PROPERTY

PROPERTY ErrorIndex : reference to uint
SET
_nErrIndex  REF= ErrorIndex;
END_SET
END_PROPERTY

PROPERTY FileRoot : pointer to string(255)
SET
_pFileRoot := FileRoot;
END_SET
END_PROPERTY

METHOD FolderDate : STRING
VAR_INPUT
	LocalTime   : POINTER TO DT;
END_VAR
VAR
	sTmp        : STRING;
END_VAR
IF NOT (LocalTime <> 0)
THEN
	FolderDate := 'NULL';
	RETURN;
END_IF

sTmp := DT_TO_STRING(LocalTime^);

// cut off #dt literal
sTmp := right(sTmp, len(sTmp)-3);

sTmp := replace(sTmp, '_', 1, 5);
sTmp := replace(sTmp, '_', 1, 8);

sTmp := left(sTmp,10);	// year_month_day

FolderDate := sTmp;
END_METHOD

PROPERTY LocalTime : pointer to DT
SET
_dtLocalTime := LocalTime;
END_SET
END_PROPERTY

PROPERTY MessageIndex : reference to uint
SET
_nMsgIndex   REF= MessageIndex;
END_SET
END_PROPERTY

PROPERTY MsgList : pointer to ARRAY[1..GVL_MSG.MAX_MESSAGE] OF st_message
SET
_pMsgList := MsgList;
END_SET
END_PROPERTY

METHOD StringLen : UINT // 	string length for len > 255
VAR_INPUT
  pInString		: POINTER TO STRING(STR_LEN);
END_VAR
VAR
	Counter			: UINT;
	pInWork			: POINTER TO BYTE;
END_VAR
pInWork := pInString;
Counter := 0;

WHILE (pInWork^ <> 0) AND
			(Counter < STR_LEN)
DO
	Counter := Counter + 1;
	pInWork := pInWork + 1;
END_WHILE

StringLen := Counter;
END_METHOD

METHOD WriteData  : e_progress
VAR_INPUT
  bExecute        : BOOL;
END_VAR
VAR_INST
  _eState         : e_progress;
  _bError         : BOOL;
  _nErrorId       : UDINT;
END_VAR
IF NOT bExecute
THEN
  _eState                     := E_PROGRESS.PROGRESS_INIT;
END_IF

CASE _eState 
OF

	E_PROGRESS.PROGRESS_INIT:
		_fbFileOpen.bExecute      := FALSE;
		_fbFileWrite.bExecute	    := FALSE;
		_fbFileClose.bExecute	    := FALSE;

		IF bExecute
		THEN
      _nErrorId               := 0;
      _eState                 := E_PROGRESS.PROGRESS_BUSY;
		END_IF

	E_PROGRESS.PROGRESS_BUSY:
		_fbFileOpen.bExecute      := TRUE;

    IF _fbFileOpen.bError
    THEN
		  _fbFileOpen.bExecute    := FALSE;
      _nErrorId               := _fbFileOpen.nErrId;
      _eState                 := E_PROGRESS.PROGRESS_ERROR;

		ELSIF _fbFileOpen.bBusy
		THEN
      _eState                 := E_PROGRESS.PROGRESS_PREPARE;
		END_IF

	E_PROGRESS.PROGRESS_PREPARE:
		IF NOT _fbFileOpen.bBusy
		THEN
		  _fbFileOpen.bExecute    := FALSE;
			_fbFileWrite.bExecute   := TRUE;
      _eState                 := E_PROGRESS.PROGRESS_STARTUP;
		END_IF

	E_PROGRESS.PROGRESS_STARTUP:
    IF _fbFileWrite.bError
    THEN
			_fbFileWrite.bExecute   := FALSE;
      _nErrorId               := _fbFileWrite.nErrId;
      _eState                 := E_PROGRESS.PROGRESS_ERROR;

		ELSIF _fbFileWrite.bBusy
		THEN
      _eState                 := E_PROGRESS.PROGRESS_CHECK;
		END_IF

	E_PROGRESS.PROGRESS_CHECK:
		IF NOT _fbFileWrite.bBusy
		THEN
			_fbFileWrite.bExecute   := FALSE;
			_fbFileClose.bExecute   := TRUE;
      _eState                 := E_PROGRESS.PROGRESS_OCCUPIED;
		END_IF

	E_PROGRESS.PROGRESS_OCCUPIED:
    IF _fbFileClose.bError
    THEN
			_fbFileClose.bExecute   := FALSE;
      _nErrorId               := _fbFileClose.nErrId;
      _eState                 := E_PROGRESS.PROGRESS_ERROR;

		ELSIF _fbFileClose.bBusy
		THEN
      _eState                 := E_PROGRESS.PROGRESS_WORKING;
		END_IF

	E_PROGRESS.PROGRESS_WORKING:
		IF NOT _fbFileClose.bBusy
		THEN
			_fbFileClose.bExecute   := FALSE;
      _eState                 := E_PROGRESS.PROGRESS_DONE;
		END_IF
END_CASE


_fbFileOpen(
	sNetId:= , 
	sPathName:= _sFilename, 
	nMode:= FOPEN_MODEAPPEND OR FOPEN_MODEPLUS, 
	ePath:= PATH_GENERIC, 
	bExecute:= , 
	tTimeout:= T#10S, 
	bBusy=> , 
	bError=> , 
	nErrId=> , 
	hFile=> );

_fbFileWrite(
	sNetId:= , 
	hFile:= _fbFileOpen.hFile, 
	pWriteBuff:= ADR(_sWriteData), 
	cbWriteLen:= StringLen(ADR(_sWriteData)), 
	bExecute:= , 
	tTimeout:= T#10S, 
	bBusy=> , 
	bError=> , 
	nErrId=> , 
	cbWrite=> );

_fbFileClose(
	sNetId:= , 
	hFile:= _fbFileOpen.hFile, 
	bExecute:= , 
	tTimeout:= T#10S, 
	bBusy=> , 
	bError=> , 
	nErrId=> );

WriteData                     := _eState;
END_METHOD

END_FUNCTION_BLOCK

// ---- XTS/_Visualization/GROUP_VISU.TcVIS
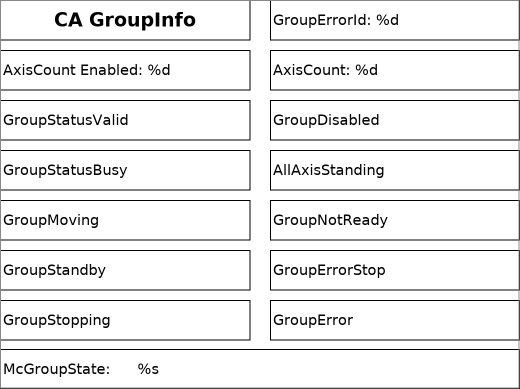
VISUALIZATION GROUP_VISU  // 520x389
VAR_IN_OUT
	stGroupInfo   : ST_GROUP_INFO;
  sGroupState   : string(60);
END_VAR
    Rectangle (0,100 250x40), "GroupStatusValid", colour toggle: stGroupInfo.GroupStatusValid
    Rectangle (0,150 250x40), "GroupStatusBusy", colour toggle: stGroupInfo.GroupStatusBusy
    Rectangle (0,200 250x40), "GroupMoving", colour toggle: stGroupInfo.GroupMoving
    Rectangle (270,250 250x40), "GroupErrorStop", colour toggle: stGroupInfo.GroupErrorStop
    Rectangle (270,200 250x40), "GroupNotReady", colour toggle: stGroupInfo.GroupNotReady
    Rectangle (0,250 250x40), "GroupStandby", colour toggle: stGroupInfo.GroupStandby
    Rectangle (0,300 250x40), "GroupStopping", colour toggle: stGroupInfo.GroupStopping
    Rectangle (270,100 250x40), "GroupDisabled", colour toggle: stGroupInfo.GroupDisabled
    Rectangle (270,150 250x40), "AllAxisStanding", colour toggle: stGroupInfo.AllAxesStanding
    Rectangle (270,300 250x40), "GroupError", colour toggle: stGroupInfo.GroupError
    Rectangle (270,0 250x40), "GroupErrorId: %d", text variable: stGroupInfo.GroupErrorId
    Rectangle (270,50 250x40), "AxisCount: %d", text variable: stGroupInfo.AxisCount
    Rectangle (0,349 520x40), "McGroupState: %s", text variable: sGroupState
    Rectangle (0,0 250x40), "CA GroupInfo"
    Rectangle (0,50 250x40), "AxisCount Enabled: %d", text variable: stGroupInfo.AxisCountEnabled
END_VISUALIZATION

// ---- XTS/_Visualization/textlists/TL_E_CTRL_MOVER.TcTLO
TEXTLIST TL_E_CTRL_MOVER
  0 = 'MOVER_NULL'
  1 = 'MOVER_ENABLE'
  2 = 'MOVER_DISABLE'
  4 = 'MOVER_MOVE_TO_POS_CA'
  5 = 'MOVER_SEND_TO_POS_CA'
  6 = 'MOVER_HALT'
  7 = 'MOVER_GEAR_IN'
  8 = 'MOVER_GEAR_IN_POS_CA'
  9 = 'MOVER_GEAR_OUT'
  10 = 'MOVER_RESET'
  3 = 'MOVER_MOVE_TO_POS'
  11 = 'MOVER_MOVE_TO_POS_ABS'
   = ''
END_TEXTLIST
